// TIA Portal V19 export
FUNCTION "FC_Pomiar" : Void   // FC2, LAD
{ S7_Optimized_Access := 'TRUE' }
// stored: SetENOAutomatically false
BEGIN
END_FUNCTION
